(* IEC 61131-3 sources: Yaha/Documentation/Infomaterial/OSCAT/pcworx_building_100/pcworx_building_100/pcworx_building_100_module_export (part 2) *)

(* ---- TEMP_EXT.ST ---- *)
(*@PROPERTIES_EX@
TYPE: POU
LOCALE: 0
IEC_LANGUAGE: ST
PLC_TYPE: independent
PROC_TYPE: independent
GROUP: HLK
*)
(*@KEY@:DESCRIPTION*)
version 1.3	13. mar. 2009
programmer 	hugo
tested by	oscat

temp_ext measures and processes ext temperature and decides if heating or cooling is needed.

 the measurement of t_ext has 3 inputs which can be configured in different ways:
	t_ext_config = 0 means the ext temp is the avg of the 3 external temperatures, this mode is the default mode.
	t_ext_config = 1 means t_ext1 is used.
	t_ext_config = 2 means t_ext1 is used.
	t_ext_config = 3 means t_ext1 is used.
	t_ext_config = 4 means t_ext_default is used.
	t_ext_config = 5 means the lowest of the 3 external temperatures is used.
	t_ext_config = 6 means the higest externnal temperature is used.
	t_ext_config = 7 means the midlle external temperature is used, if there are only two working, the lowest is used.
	in any config mode, an external temperature higher then t_ext_max or lower then t_ext_min is ignored to prevent from temperatures caused by broken sensors or wires.
	if no external temperature is available, a default value (t_ext_default) is used.
	if you have only one external sensor, connect the 3 inputs to the same sensor, or select the right input with t_ext_config.

heating or cooling is enabled during heating / cooling period when the day or night start temperature is reached for at least the specified delay time and will be disabled after the stop temperature is reached.
t_ext output can be used by other modules to determine the correct system temperature for heating or cooling.
(*@KEY@:END_DESCRIPTION*)
FUNCTION_BLOCK TEMP_EXT

(*Group:Default*)

VAR_INPUT
	T_EXT1 :	REAL;
	T_EXT2 :	REAL;
	T_EXT3 :	REAL;
	T_EXT_CONFIG :	BYTE := 0;
	DT_IN :	UDINT;
	T_EXT_MIN :	REAL := REAL#-40.0;
	T_EXT_MAX :	REAL := REAL#60.0;
	T_EXT_DEFAULT :	REAL := REAL#-10.0;
	HEAT_PERIOD_START :	UDINT := UDINT#20995200;(*Anfangswert: D#1970-9-1*)
	HEAT_PERIOD_STOP :	UDINT := UDINT#10281600;(*Anfangswert: D#1970-4-30*)
	COOL_PERIOD_START :	UDINT := UDINT#07776000;(*Anfangswert: D#1970-4-1*)
	COOL_PERIOD_STOP :	UDINT := UDINT#23500800;(*Anfangswert: D#1970-9-30*)
	HEAT_START_TEMP_DAY :	REAL := REAL#15.0;
	HEAT_START_TEMP_NIGHT :	REAL := REAL#10.0;
	HEAT_STOP_TEMP :	REAL := REAL#18.0;
	COOL_START_TEMP_DAY :	REAL := REAL#26.0;
	COOL_START_TEMP_NIGHT :	REAL := REAL#26.0;
	COOL_STOP_TEMP :	REAL := REAL#24.0;
	START_DAY :	UDINT := UDINT#32400000;(*Anfangswert:TOD#09:00*)
	START_NIGHT :	UDINT := UDINT#75600000;(*Anfangswert:TOD#21:00*)
	CYCLE_TIME :	TIME := t#10m;
END_VAR

VAR_OUTPUT
	T_EXT :	REAL;
	HEAT :	BOOL;
	COOL :	BOOL;
END_VAR

VAR
	tx :	TIME;
	last_run :	TIME;
	init :	BOOL;
	cool_start :	UDINT;
	cool_stop :	UDINT;
	heat_start :	UDINT;
	heat_stop :	UDINT;
	xdate :	UDINT;
	day :	BOOL;
	T_PLC_MS :	T_PLC_MS;
END_VAR

(*@KEY@: WORKSHEET
NAME: TEMP_EXT
IEC_LANGUAGE: ST
*)
IF NOT init THEN
	init := TRUE;
	heat_start := SET_DATE(1972,MONTH_OF_DATE(heat_period_start),DAY_OF_MONTH(heat_period_start));
	heat_stop := SET_DATE(1972,MONTH_OF_DATE(heat_period_stop),DAY_OF_MONTH(heat_period_stop));
	cool_start := SET_DATE(1972,MONTH_OF_DATE(cool_period_start),DAY_OF_MONTH(cool_period_start));
	cool_stop := SET_DATE(1972,MONTH_OF_DATE(cool_period_stop),DAY_OF_MONTH(cool_period_stop));
END_IF;

(* read system time *)
T_PLC_MS();
tx:= UDINT_TO_TIME(T_PLC_MS.T_PLC_MS);

(* for efficiency exit isf this program has been executed less then 1min ago *)
IF tx - last_run < cycle_time THEN RETURN; END_IF;

(* calculate frequently used variables *)
xdate := SET_DATE(1972,MONTH_OF_DATE(DT_TO_DATE(dt_in)),DAY_OF_MONTH(DT_TO_DATE(dt_in)));
day := DT_TO_TOD(dt_in) >= start_day AND  DT_TO_TOD(dt_in) < start_night;

(* read the correct external temperature depending on the t_ext_config setting *)
t_ext := MULTI_IN(t_ext1, t_ext2, t_ext3, t_ext_default, t_ext_min, t_ext_max, t_ext_config);

(* dtermine heating *)
IF (heat_start <= heat_stop AND xdate >= heat_start AND xdate <= heat_stop) OR (heat_start > heat_stop AND (xdate >= heat_start OR xdate <= heat_stop)) THEN
	(* heating period id true check for temperature *)
	IF day AND t_ext <= heat_start_temp_day THEN
		heat := TRUE;
	ELSIF NOT day AND t_ext <= heat_start_temp_night THEN
		heat := TRUE;
	ELSIF t_ext >= heat_stop_temp THEN
		heat := FALSE;
	END_IF;
ELSE
	heat := FALSE;
END_IF;

(* dtermine cooling *)
IF (cool_start <= cool_stop AND xdate >= cool_start AND xdate <= cool_stop) OR (cool_start > cool_stop AND (xdate >= cool_start OR xdate <= cool_stop)) THEN
	(* cooling period is true check for temperature *)
	IF day AND t_ext >= cool_start_temp_day THEN
		cool := TRUE;
	ELSIF NOT day AND t_ext >= cool_start_temp_night THEN
		cool := TRUE;
	ELSIF t_ext <= cool_stop_temp THEN
		cool := FALSE;
	END_IF;
ELSE
	cool := FALSE;
END_IF;

last_run := tx;

(* revision history
hm	6 dec 2006	rev 1.0
	original version

hm	15.9.2007		rev 1.1
	replaced Time() with T_PLC_MS for compatibility and performance reasons

hm	7. oct. 2008	rev 1.2
	changed name of function month to month_of_date

hm	13. mar. 2009	rev 1.3
	real constants updated to new systax using dot

*)
(*@KEY@: END_WORKSHEET *)
END_FUNCTION_BLOCK

(* ---- TIMER_1.ST ---- *)
(*@PROPERTIES_EX@
TYPE: POU
LOCALE: 0
IEC_LANGUAGE: ST
PLC_TYPE: independent
PROC_TYPE: independent
GROUP: ELECTRICAL
*)
(*@KEY@:DESCRIPTION*)
version 2.2	16. dec. 2009
programmer 	oscat
tested by	oscat

this is a simple timer that generates an output pulse on selected days.
the output pulse width can be programmed with duration, if set to 0 no pulse is generated.
day specifies the specific days for the event to occur, bit 0 = sunday, bit 1 = saturday, bit 2 = friday ....
for all days to be active 127 has to be specified for DAY.
(*@KEY@:END_DESCRIPTION*)
FUNCTION_BLOCK TIMER_1

(*Group:Default*)

VAR_INPUT
	E :	BOOL := TRUE;
	DTI :	UDINT;
	START :	UDINT;
	DURATION :	TIME;
	DAY :	BYTE := BYTE#2#0111_1111;
END_VAR

VAR_OUTPUT
	Q :	BOOL;
	STOP :	TIME;
END_VAR

(*@KEY@: WORKSHEET
NAME: TIMER_1
IEC_LANGUAGE: ST
*)
IF E THEN
	stop := TOD_TO_TIME(START) + DURATION;
	IF stop > T#24h THEN stop := stop - T#24h; END_IF;
	Q := TIMECHECK(DT_TO_TOD(DTI), START, TIME_TO_TOD(stop)) AND (SHR(BYTE#128, DAY_OF_WEEK(DT_TO_DATE(DTI))) AND DAY) > BYTE#0;
ELSE
	Q := FALSE; (* clear output when e is not true *)
END_IF;

(*
1.12.2006 hm		rev 1.1
	corrected an error with pulse width = 0.

25.12.2006 hm		rev 1.2
	corrected an error when timer overflows.

14.apr 2007 hm		rev 1.3
	corrected an error while while output would not go active when start year would be 1970.
	increase accuracy by checking every 100ms
	added init section to compensate for timer overflow

15.9.2007 hm		rev 1.4
	replaced Time() with T_PLC_MS for compatibility and performance reasons

hm	1. okt 2007		rev 1.5
	corrected an error while output would not stay active over midnight.

hm	17. jan 2008	rev 1.6
	New code with better performance
	Output is now only active during the time of day it is supposed to
	no pulse is generated at power up

hm	7. oct. 2008	rev 1.7
	changed function weekday to day_of_week

hm	23. oct. 2008	rev 2.0
	new code, added input E, now days can be selected by bits in byte day

hm	6. nov. 2008	rev 2.1
	added default for input EN and input DAY

hm 16. dec 2009	rev 2.2
	fixed a bug over midnight

*)
(*@KEY@: END_WORKSHEET *)
END_FUNCTION_BLOCK

(* ---- TIMER_2.ST ---- *)
(*@PROPERTIES_EX@
TYPE: POU
LOCALE: 0
IEC_LANGUAGE: ST
PLC_TYPE: independent
PROC_TYPE: independent
GROUP: ELECTRICAL
*)
(*@KEY@:DESCRIPTION*)
version 1.5	22.dec.2008
programmer 	oscat
tested by	oscat

this timer generated programmabe output pulses per day, week, month and so on.
the mode input determines on which days the timer will be active.
	mode = 0			never
	mode = 1..7			monday .. sunday
	mode = 11			every day
	mode = 12			every second day
	mode = 13			every 3rd day
	mode = 14			every 4th day
	mode = 15			every 5th day
	mode = 16 			every 6th day
	mode = 20			only monday - friday
	mode = 21			only sat - sunday
	mode = 22			workdays only
	mode = 23			holidays and weekend
	mode = 24			holidays only
	mode = 25			every 1st day of the month
	mode = 26			every last day of the month
	mode = 27			every 31 of december
	mode = 28			every 1st of january

a holiday input can be used to supply holiday information to the module.
(*@KEY@:END_DESCRIPTION*)
FUNCTION_BLOCK TIMER_2

(*Group:Default*)

VAR_INPUT
	DT_IN :	UDINT;
	START :	UDINT;
	DURATION :	TIME;
	MODE :	BYTE;
	HOLIDAY :	BOOL;
END_VAR

VAR_OUTPUT
	Q :	BOOL;
END_VAR

VAR
	last_check :	TIME := T#0s;
	dat :	UDINT;
	daytime :	UDINT;
	activation :	TIME;
	tx :	TIME;
	enabled :	BOOL;
	wday :	INT;
	init :	BOOL;
END_VAR

VAR RETAIN
	run_date :	UDINT;
END_VAR

VAR
	T_PLC_MS :	T_PLC_MS;
END_VAR

(*@KEY@: WORKSHEET
NAME: TIMER_2
IEC_LANGUAGE: ST
*)
(* read system time *)
T_PLC_MS();
tx:= UDINT_TO_TIME(T_PLC_MS.T_PLC_MS);

IF NOT init THEN
	init := TRUE;
	last_check := tx - t#100ms;
END_IF;

(* for performance resons exit if execution is not necessary *)
IF tx - last_check < T#100ms THEN RETURN; END_IF;

(* calculate temp variables *)
dat := DT_TO_DATE(dt_in);
daytime := DT_TO_TOD(dt_in);
wday := DAY_OF_WEEK(dat);

(* calculate if any action is necessary today *)
CASE _BYTE_TO_INT(mode) OF
1..7:	(* mondays to fridays *)
	enabled := wday = _BYTE_TO_INT(mode);
11:	(* every day *)
	enabled := TRUE;
12..16:	(* every nth day *)
	enabled := (dat / UDINT#86400) MOD (BYTE_TO_UDINT(mode) - UDINT#10) = UDINT#0;
20:	(* monday - friday *)
	enabled := wday <= 5;
21:	(* saturday and sunday *)
	enabled := wday > 5;
22: (* workdays only *)
	enabled := wday <= 5 AND NOT holiday;
23:	(* holidays and weekends *)
	enabled := wday > 5 OR holiday;
24:	(* holidays only *)
	enabled := holiday;
25:	(* 1st day of the month *)
	enabled := DAY_OF_MONTH(dat) = 1;
26:	(* last day of month *)
	enabled := day_of_month(dat + TIME_TO_UDINT(t#1d)) = 1;
27:	(* 31st of december *)
	enabled := DAY_OF_MONTH(dat) = 31 AND MONTH_OF_DATE(dat) = 12;
28:	(* 1st of january *)
	enabled := DAY_OF_YEAR(dat) = 1;
ELSE
	enabled := FALSE;
END_CASE;

(* set output if necessary *)
IF enabled AND NOT Q AND daytime >= start AND run_date <> dat THEN
	Q := TRUE;
	activation := tx;
	run_date := dat;
ELSIF Q AND tx - activation >= duration THEN
	Q := FALSE;
END_IF;
last_check := Tx;

(* revision history
hm 22.2.2007		rev 1.1
	changed VAR RETAIN PERSISTENT to VAR RETAIN for better compatibility
	wago lon contollers do not support persisitent

hm	15.9.2007		rev 1.2
	replaced Time() with T_PLC_MS for compatibility and performance reasons

hm	7. oct. 2008	rev 1.3
	changed function month to month_of_date

hm	20. oct. 2008	rev 1.4
	improved performance
	deleted unnecessary trunc

hm	22. dec. 2008	rev 1.5
	make sure timer_2 is executed in the first cycle

*)
(*@KEY@: END_WORKSHEET *)
END_FUNCTION_BLOCK

(* ---- TIMER_EVENT_DECODE.ST ---- *)
(*@PROPERTIES_EX@
TYPE: POU
LOCALE: 0
IEC_LANGUAGE: ST
PLC_TYPE: independent
PROC_TYPE: independent
GROUP: ELECTRICAL
*)
(*@KEY@:DESCRIPTION*)
version 1.1	25. oct. 2008
programmer 	hugo
tested by	oscat

STRING_TO_TIMER_EVENT converts a string to a timer event structure.
(*@KEY@:END_DESCRIPTION*)
FUNCTION_BLOCK TIMER_EVENT_DECODE

(*Group:Default*)

VAR_INPUT
	EVENT :	oscat_STRING250;
	LANG :	INT;
END_VAR

VAR_OUTPUT
	TIMER_EVENT_DECODE :	oscat_TIMER_EVENT_DATA;
END_VAR

VAR
	pos :	INT;
	start :	INT;
	stop :	INT;
	step :	INT;
	tmp :	oscat_STRING60;
	char :	INT;
	FSTRING_TO_BYTE :	FSTRING_TO_BYTE;
	IS_CC :	IS_CC;
	FSTRING_TO_WEEK :	FSTRING_TO_WEEK;
	FSTRING_TO_WEEKDAY :	FSTRING_TO_WEEKDAY;
	STRING_TO_TOD :	STRING_TO_TOD;
	_STRING_TO_TIME :	_STRING_TO_TIME;
END_VAR

(*@KEY@: WORKSHEET
NAME: TIMER_EVENT_DECODE
IEC_LANGUAGE: ST
*)
(* a timer event is specified as follows:
	$typ;ch;day;start;duration;land;lor#
$ 		= start of definition
typ 	= type of definition	(number)
channel	= channel number		(number)
day 	= day number			(number)
start	= start time			(time of day)
duration= duration of event		(time)
land	= mask for output AND	(8bit value)
lor		= mask for ourput OR	(8bit value)
#		= end of definition
*)

(* check for start and ending character *)
stop := LEN(event);
IF (GET_CHAR(event,1) <> 60) AND (GET_CHAR(event,stop) <> 62) THEN RETURN; END_IF;
start := 2;
step := 0;

(* parse the string for next ; *)
FOR pos := 2 TO stop DO
    char := GET_CHAR(event,pos);

	IF char = 59 OR char = 62 THEN
		tmp := MID(event, pos - start, start);
		CASE step OF
			0:	(* read type *)
                FSTRING_TO_BYTE(IN:=tmp);
                TIMER_EVENT_DECODE.typ := FSTRING_TO_BYTE.FSTRING_TO_BYTE;

			1:	(* read channel *)
                FSTRING_TO_BYTE(IN:=tmp);
                TIMER_EVENT_DECODE.channel := FSTRING_TO_BYTE.FSTRING_TO_BYTE;

			2:	(* read day *)
                IS_CC(str:=tmp,cmp:='0123456789abcdefABCDEF#');

				IF IS_CC.IS_CC THEN
                    FSTRING_TO_BYTE(IN:=tmp);
                    TIMER_EVENT_DECODE.DAY := FSTRING_TO_BYTE.FSTRING_TO_BYTE;
				ELSIF TIMER_EVENT_DECODE.typ = BYTE#2 THEN
                    FSTRING_TO_WEEK(WEEK:=tmp,LANG:=LANG);
                    TIMER_EVENT_DECODE.DAY := FSTRING_TO_WEEK.FSTRING_TO_WEEK;
				ELSE
                    FSTRING_TO_WEEKDAY(WDAY:=tmp,LANG:=LANG);
                    TIMER_EVENT_DECODE.DAY := INT_TO_BYTE(FSTRING_TO_WEEKDAY.FSTRING_TO_WEEKDAY);
				END_IF;

			3:	(* read start *)
			    STRING_TO_TOD(_TOD:=tmp);
                TIMER_EVENT_DECODE.start := STRING_TO_TOD.STRING_TO_TOD;

			4:	(* read duaration *)
                _STRING_TO_TIME(_TIME:=tmp);
                TIMER_EVENT_DECODE.duration := _STRING_TO_TIME.STRING_TO_TIME;

			5:	(* read land *)
                FSTRING_TO_BYTE(IN:=tmp);
				TIMER_EVENT_DECODE.land := FSTRING_TO_BYTE.FSTRING_TO_BYTE;

			6:	(* read lor *)
                FSTRING_TO_BYTE(IN:=tmp);
				TIMER_EVENT_DECODE.LOR := FSTRING_TO_BYTE.FSTRING_TO_BYTE;
		END_CASE;
		start := pos + 1;
		step := step + 1;
	END_IF;
END_FOR;

(* revision history
hm	17. jun 2008	rev 1.0
	original version

hm	25. oct. 2008	rev 1.1
	adding input lang for language selection
*)
(*@KEY@: END_WORKSHEET *)
END_FUNCTION_BLOCK

(* ---- TIMER_EXT.ST ---- *)
(*@PROPERTIES_EX@
TYPE: POU
LOCALE: 0
IEC_LANGUAGE: ST
PLC_TYPE: independent
PROC_TYPE: independent
GROUP: ELECTRICAL
*)
(*@KEY@:DESCRIPTION*)
version 1.0	7. oct. 2008
programmer 	oscat
tested by	tobias

TIMER_EXT is a twilight timer.
the timer can be programmed to switch lights or other equippment or during twilight times.
in addition to the automatik mode the timer can be stopped and started by a switch at any given time.
An enable input ENA can be used for external control.
two inputs ON and OFF can be used to statically control the output.
the timer can be programmed to work on saturdays, sundays and holidays if required.
(*@KEY@:END_DESCRIPTION*)
FUNCTION_BLOCK TIMER_EXT

(*Group:Default*)

VAR_INPUT
	ENA :	BOOL;
	ON :	BOOL;
	OFF :	BOOL;
	MAN :	BOOL;
	SWITCH :	BOOL;
	DT_IN :	UDINT;
	SUN_SET :	UDINT;
	SUN_RISE :	UDINT;
	HOLIDAY :	BOOL;
	T_DEBOUNCE :	TIME := T#100ms;
	T_RISE_START :	TIME;
	T_RISE_STOP :	TIME;
	T_SET_START :	TIME;
	T_SET_STOP :	TIME;
	T_DAY_START :	UDINT;
	T_DAY_STOP :	UDINT;
	ENABLE_SATURDAY :	BOOL;
	ENABLE_SUNDAY :	BOOL;
	ENABLE_HOLIDAY :	BOOL;
END_VAR

VAR_OUTPUT
	Q :	BOOL;
	STATUS :	BYTE;
END_VAR

VAR
	mx :	MANUAL_2;
	deb :	DEBOUNCE;
	tdx :	UDINT;
	wdx :	INT;
	tc :	TIME;
	tx :	UDINT;
	tl :	UDINT;
	qx :	BOOL;
	T_PLC_MS :	T_PLC_MS;
	init :	BOOL;
END_VAR

(*@KEY@: WORKSHEET
NAME: TIMER_EXT
IEC_LANGUAGE: ST
*)
(* lösche die millisekunden bei sunrise und sunset *)
SUN_RISE := SUN_RISE / UDINT#1000 * UDINT#1000;
SUN_SET := SUN_SET / UDINT#1000 * UDINT#1000;

(* measure cycle time tc and make sure this circuitry is not called more then once in 200ms*)
T_PLC_MS();
tx:= T_PLC_MS.T_PLC_MS;
IF NOT init THEN
	init := TRUE;
	tl := tx;
END_IF;
tc := UDINT_TO_TIME(tx - tl);
IF tc < t#200ms THEN RETURN; END_IF;
tl := tx;

(* debounce *)
deb(in := SWITCH, TD := T_DEBOUNCE, PM := TRUE);

(* read time of day and strip off all milliseconds *)
tdx := DT_TO_TOD(dt_in);
wdx := DAY_OF_WEEK(DT_TO_DATE(dt_in));

(* automatic output control *)
IF deb.Q THEN
	qx := NOT qx;
	status := BYTE#110;
ELSIF holiday AND NOT enable_holiday THEN
	qx := FALSE;
ELSIF wdx = 6 AND NOT enable_saturday THEN
	qx := FALSE;
ELSIF wdx = 7 AND NOT enable_sunday THEN
	qx := FALSE;
ELSIF T_day_start > UDINT#00 (* TOD#00:00 *) AND tdx - T_DAY_START <= TIME_TO_UDINT(tc) THEN
	(* turn on at specified daytime *)
	qx := TRUE;
	status := BYTE#111;
ELSIF T_DAY_STOP > UDINT#00 (* TOD#00:00 *) AND tdx - T_DAY_STOP <= TIME_TO_UDINT(tc) THEN
	(* turn off at specific daytime *)
	qx := FALSE;
	status := BYTE#112;
ELSIF T_RISE_START > T#0s AND tdx - SUN_RISE + TIME_TO_UDINT(T_RISE_START) <= TIME_TO_UDINT(tc) THEN
	(* turn on before sunrise *)
	qx := TRUE;
	status := BYTE#113;
ELSIF T_RISE_STOP > T#0s AND tdx - SUN_RISE - TIME_TO_UDINT(T_RISE_STOP) <= TIME_TO_UDINT(tc) THEN
	(* turn off after sunrise *)
	qx := FALSE;
	status := BYTE#114;
ELSIF T_SET_start > T#0s AND tdx - SUN_SET + TIME_TO_UDINT(T_SET_START) <= TIME_TO_UDINT(tc) THEN
	(* turn on before sunset *)
	qx := TRUE;
	status := BYTE#115;
ELSIF T_SET_STOP > T#0s AND tdx - SUN_SET - TIME_TO_UDINT(T_SET_STOP) <= TIME_TO_UDINT(tc) THEN
	(* turn off after sunset *)
	qx := FALSE;
	status := BYTE#116;
END_IF;

(* manual and output control *)
mx(in := qx, ena := ENA, on := ON, off := OFF, man := MAN);
Q := mx.Q;

(* set the status output *)
IF mx.STATUS > BYTE#100 THEN status := mx.STATUS; END_IF;

(*
hm 7. oct. 2008	rev 1.0
	original version

*)
(*@KEY@: END_WORKSHEET *)
END_FUNCTION_BLOCK

(* ---- TIMER_P4.ST ---- *)
(*@PROPERTIES_EX@
TYPE: POU
LOCALE: 0
IEC_LANGUAGE: ST
PLC_TYPE: independent
PROC_TYPE: independent
GROUP: ELECTRICAL
*)
(*@KEY@:DESCRIPTION*)
version 1.4	26. jan. 2011
programmer 	hugo
tested by	oscat

TIMER_P4 is a programmable universal timer.
(*@KEY@:END_DESCRIPTION*)
FUNCTION_BLOCK TIMER_P4

(*Group:Default*)

VAR_INPUT
	DTIME :	UDINT;
	TREF_0 :	UDINT;
	TREF_1 :	UDINT;
	HOLY :	BOOL;
	L0 :	BOOL;
	L1 :	BOOL;
	L2 :	BOOL;
	L3 :	BOOL;
	OFS :	BYTE;
	ENQ :	BOOL;
	MAN :	BOOL;
	MI :	BYTE;
	RST :	BOOL;
END_VAR

VAR_IN_OUT
	PROG :	oscat_TIMER_EVENT;
END_VAR

VAR_OUTPUT
	Q0 :	BOOL;
	Q1 :	BOOL;
	Q2 :	BOOL;
	Q3 :	BOOL;
	STATUS :	BYTE;
END_VAR

VAR
	day_start :	UDINT;
	start :	UDINT;
	event :	oscat_TIMER_EVENT_DATA;
	pos :	INT;
	last_execute :	UDINT;
	current_day :	DINT;
	mask :	BYTE;
	ma :	oscat_arb_0_3;
	mo :	oscat_arb_0_3;
	qn :	oscat_TP4_qn;
	qs :	oscat_TP4_qn;
	channel :	INT;
	tx :	UDINT;
	array_max :	INT := 63;
	channel_max :	INT := 3;
END_VAR

(*@KEY@: WORKSHEET
NAME: TIMER_P4
IEC_LANGUAGE: ST
*)
(* for performance reasons we only execute the code at the beginning of a new second *)

IF RST THEN
	(* reset all events to last active on 1.1.1970 *)
	last_execute := UDINT#00; (* DT#1970-1-1-00:00 *)
	FOR pos := 0 TO ARRAY_MAX DO
		IF (PROG[pos].CHANNEL >= OFS) AND (_BYTE_TO_INT(PROG[pos].CHANNEL) < (_BYTE_TO_INT(OFS) + 4)) THEN PROG[pos].LAST := last_execute; END_IF;
	END_FOR;

	(* reset all set markers and logic masks *)
	FOR pos := 0 TO channel_max DO
		qs[pos] := FALSE;
	END_FOR;

(* normal operation *)
ELSIF dtime <> last_execute THEN
	(* save the actual second for next execution test *)
	last_execute := DTIME;

	(* calculate dt for the start of the day to be used in comparisons *)
	day_start := DATE_TO_DT(DT_TO_DATE(DTIME));

	(* set all qn to FALSE *)
	FOR pos := 0 TO channel_max DO qn[pos] := FALSE; END_FOR;

	(* search the array PROG for timer events *)
	FOR pos := 0 TO ARRAY_MAX DO
		event := prog[pos];
		channel := _BYTE_TO_INT(event.CHANNEL) - _BYTE_TO_INT(OFS);
		IF (event.TYP > BYTE#0) AND (channel >= 0) AND (channel <= channel_max) THEN
			ma[channel] := event.LAND;
			mo[channel] := event.LOR;
			CASE _BYTE_TO_INT(event.TYP) OF
				1:	(* daily event *)
					start := day_start + event.start;
					qn[channel] := dtime >= start AND dtime <= start + TIME_TO_UDINT(event.DURATION);

				2: 	(* event by selected weekdays *)
					IF (SHR(BYTE#128, DAY_OF_WEEK(DT_TO_DATE(Dtime))) AND event.DAY) > BYTE#0 THEN
						start := day_start + event.start;
						qn[channel] := dtime >= start AND dtime <= start + TIME_TO_UDINT(event.DURATION);
					END_IF;

				3:	(* event every N days *)
					IF current_day MOD _BYTE_TO_DINT(event.DAY) = DINT#0 THEN
						start := day_start + event.start;
						qn[channel] := dtime >= start AND dtime <= start + TIME_TO_UDINT(event.DURATION);
					END_IF;

				10:	(* weekly event exactly once a week the weekday is specified in day, 1= mo *)
					IF DAY_OF_WEEK(DT_TO_DATE(DTIME)) = BYTE_TO_INT(event.DAY) THEN
						start := day_start + event.start;
						qn[channel] := dtime >= start AND dtime <= start + TIME_TO_UDINT(event.DURATION);
					END_IF;

				20:	(* monthly event *)
					IF DAY_OF_MONTH(DT_TO_DATE(DTIME)) = BYTE_TO_INT(event.DAY) THEN
						start := day_start + event.start;
						qn[channel] := dtime >= start AND dtime <= start + TIME_TO_UDINT(event.DURATION);
					END_IF;

				21:	(* event on last day of month *)
					IF DT_TO_DATE(DTIME) = MONTH_END(DT_TO_DATE(dtime)) THEN
						start := day_start + event.start;
						qn[channel] := dtime >= start AND dtime <= start + TIME_TO_UDINT(event.DURATION);
					END_IF;

				30:	(* yearly event on a specific day specified in day *)
					IF DAY_OF_YEAR(DT_TO_DATE(DTIME)) = BYTE_TO_INT(event.DAY) THEN
						start := day_start + event.start;
						qn[channel] := dtime >= start AND dtime <= start + TIME_TO_UDINT(event.DURATION);
					END_IF;

				31:	(* event on last day of year *)
					IF DT_TO_DATE(DTIME) = YEAR_END(YEAR_OF_DATE(DT_TO_DATE(dtime))) THEN
						start := day_start + event.start;
						qn[channel] := dtime >= start AND dtime <= start + TIME_TO_UDINT(event.DURATION);
					END_IF;

				40:	(* event on leap days *)
					IF LEAP_DAY(DT_TO_DATE(dtime)) THEN
						start := day_start + event.start;
						qn[channel] := dtime >= start AND dtime <= start + TIME_TO_UDINT(event.DURATION);
					END_IF;

				41: (* event on holidays *)
					IF HOLY THEN
						start := day_start + event.start;
						qn[channel] := dtime >= start AND dtime <= start + TIME_TO_UDINT(event.DURATION);
					END_IF;

				42: (* event on holidays and weekends *)
					IF (Holy OR (DAY_OF_WEEK(DT_TO_DATE(dtime)) = 6) OR (DAY_OF_WEEK(DT_TO_DATE(dtime)) = 7)) THEN
						start := day_start + event.start;
						qn[channel] := dtime >= start AND dtime <= start + TIME_TO_UDINT(event.DURATION);
					END_IF;

				43:	(* event on workdays Mo-FR and no holiday *)
					IF DAY_OF_WEEK(DT_TO_DATE(dtime)) < 6 THEN
						start := day_start + event.start;
						qn[channel] := dtime >= start AND dtime <= start + TIME_TO_UDINT(event.DURATION);
					END_IF;

				50: (* event after reference time *)
					CASE _BYTE_TO_INT(prog[pos].DAY) OF
						0:	tx := tref_0;
						1:	tx := tref_1;
					ELSE
						tx := UDINT#0 (* TOD#00:00 *);
					END_CASE;
					start := day_start + tx + event.start;
					qn[channel] := dtime >= start AND dtime <= start + TIME_TO_UDINT(event.DURATION);

				51:	(* event before reference time *)
					CASE _BYTE_TO_INT(prog[pos].DAY) OF
						0:	tx := tref_0;
						1:	tx := tref_1;
					ELSE
						tx := UDINT#0 (* TOD#00:00 *);
					END_CASE;
					start := day_start + tx - event.start;
					qn[channel] := dtime >= start AND dtime <= start + TIME_TO_UDINT(event.DURATION);

				52 : (* set output at specific time + offset  *)
					CASE _BYTE_TO_INT(prog[pos].DAY) OF
						0:	tx := tref_0;
						1:	tx := tref_1;
					ELSE
						tx := UDINT#0 (* TOD#00:00 *);
					END_CASE;
					start := day_start + tx + event.start;
					IF dtime >= start AND day_start > event.LAST THEN
						qs[channel] := TRUE;
						prog[pos].LAST := day_start;
					END_IF;

				53 : (* reset output at specific time + offset *)
					CASE _BYTE_TO_INT(prog[pos].DAY) OF
						0:	tx := tref_0;
						1:	tx := tref_1;
					ELSE
						tx := UDINT#0 (* TOD#00:00 *);
					END_CASE;
					start := day_start + tx + event.start;
					IF dtime >= start AND day_start > event.LAST THEN
						qs[channel] := FALSE;
						prog[pos].LAST := day_start;
					END_IF;

				54 : (* set output at specific time - offset  *)
					CASE _BYTE_TO_INT(prog[pos].DAY) OF
						0:	tx := tref_0;
						1:	tx := tref_1;
					ELSE
						tx := UDINT#0 (* TOD#00:00 *);
					END_CASE;
					start := day_start + tx - event.start;
					IF dtime >= start AND day_start > event.LAST THEN
						qs[channel] := TRUE;
						prog[pos].LAST := day_start;
					END_IF;

				55 : (* reset output at specific time - offset *)
					CASE _BYTE_TO_INT(prog[pos].DAY) OF
						0:	tx := tref_0;
						1:	tx := tref_1;
					ELSE
						tx := UDINT#0 (* TOD#00:00 *);
					END_CASE;
					start := day_start + tx - event.start;
					IF dtime >= start AND day_start > event.LAST THEN
						qs[channel] := FALSE;
						prog[pos].LAST := day_start;
					END_IF;
			END_CASE;
		END_IF;
	END_FOR;
END_IF;

(* prepare the logical input mask *)
mask := BYTE#255;
mask:=BIT_LOAD_B(mask,L0,0);
mask:=BIT_LOAD_B(mask,L1,1);
mask:=BIT_LOAD_B(mask,L2,2);
mask:=BIT_LOAD_B(mask,L3,3);

(* set the outputs *)
Q0 := ENQ AND ((qn[0] OR qs[0]) AND ((ma[0] AND mask) = ma[0]) OR ((mo[0] AND mask) > BYTE#0) OR (man AND BIT_OF_DWORD(BYTE_TO_DWORD(MI),0)));
Q1 := ENQ AND ((qn[1] OR qs[1]) AND ((ma[1] AND mask) = ma[1]) OR ((mo[1] AND mask) > BYTE#1) OR (man AND BIT_OF_DWORD(BYTE_TO_DWORD(MI),1)));
Q2 := ENQ AND ((qn[2] OR qs[2]) AND ((ma[2] AND mask) = ma[2]) OR ((mo[2] AND mask) > BYTE#2) OR (man AND BIT_OF_DWORD(BYTE_TO_DWORD(MI),2)));
Q3 := ENQ AND ((qn[3] OR qs[3]) AND ((ma[3] AND mask) = ma[3]) OR ((mo[3] AND mask) > BYTE#3) OR (man AND BIT_OF_DWORD(BYTE_TO_DWORD(MI),3)));

(* set status *)
IF NOT enq THEN
	status := BYTE#100;
ELSIF man THEN
	status := BYTE#101;
ELSE
	status := BYTE#102;
END_IF;

(* revision history
hm	17. jun 2008	rev 1.0
	original version

hm	9. oct. 2008	rev 1.1
	changed function year to year_of_date
	changed function weekday to day_of_week
	changed structure of program to be more efficient
	changed input DIS to ENQ

hm	18. oct. 2008	rev 1.2
	changed type of input OFS from int to byte
	added typecasts to avoid warnings

hm	28. feb. 2009	rev 1.3
	array was not correctly initialized

hm	26. jan 2011	rev 1.4
	changed code to allow events over midnight
*)
(*@KEY@: END_WORKSHEET *)
END_FUNCTION_BLOCK

(* ---- WATER_CP.ST ---- *)
(*@PROPERTIES_EX@
TYPE: POU
LOCALE: 0
IEC_LANGUAGE: ST
PLC_TYPE: independent
PROC_TYPE: independent
GROUP: HLK
*)
(*@KEY@:DESCRIPTION*)
version 1.2	13. mar. 2009
programmer 	hugo
tested by	tobias

water_cp calculates the specific heat capacity of liquid water from 0..100 °C
(*@KEY@:END_DESCRIPTION*)
FUNCTION_BLOCK WATER_CP

(*Group:Default*)

VAR_INPUT
	T :	REAL;
END_VAR

VAR_OUTPUT
	CAP :	REAL;
END_VAR

VAR
	Pts :	INT;
	data :	oscat_XY;
	FB_LINEAR_INT :	LINEAR_INT;
END_VAR

(*@KEY@: WORKSHEET
NAME: WATER_CP
IEC_LANGUAGE: ST
*)
IF Pts = 0 THEN
    Pts := 10;

    data[01][0] := REAL#0.0;
    data[01][1] := REAL#4.228;
    data[02][0] := REAL#05.0;
    data[02][1] := REAL#4.200;
    data[03][0] := REAL#10.0;
    data[03][1] := REAL#4.188;
    data[04][0] := REAL#15.0;
    data[04][1] := REAL#4.184;
    data[05][0] := REAL#50.0;
    data[05][1] := REAL#4.181;
    data[06][0] := REAL#60.0;
    data[06][1] := REAL#4.183;
    data[07][0] := REAL#70.0;
    data[07][1] := REAL#4.187;
    data[08][0] := REAL#80.0;
    data[08][1] := REAL#4.194;
    data[09][0] := REAL#90.0;
    data[09][1] := REAL#4.204;
    data[10][0] := REAL#100.0;
    data[10][1] := REAL#4.220;

END_IF;

FB_LINEAR_INT(X:=T,XY:=Data,Pts:=Pts);
cap:=FB_LINEAR_INT.LINEAR_INT;

(*
    °C - die Celsius-Temperatur in Grad Celsius
    v – das spezifische Volumen in Kubikdezimeter je Kilogramm dm³/kg
    h – die spezifische Enthalpie in Kilojoule je Kilogramm 	kJ/kg
    u – die spezifische Innere Energie in Kilojoule je Kilogramm 	kJ/kg
    s – die spezifische Entropie in Kilojoule je Kilogramm mal Kelvin 	kJ/(kg·K)
    cp - die spezifische Wärmekapazität bei konstantem Druck in Kilojoule je Kilogramm mal Kelvin 	kJ/(kg·K)
    Y – Volumenausdehnungskoeffizient in 10-3 durch Kelvin  10-3/K
    L – Wärmeleitfähigkeit in Milliwatt je Meter mal Kelvin  mW / (m·K)
    n – Viskosität in Mikropascal mal Sekunde uPa·s
    s ? – Oberflächenspannung in Millinewton je Meter  mN/m

°C 		v 				h 			u 		s 			cp 		Y 		L		n		s
-20		1,006580
0 		1,000160 		0,06 		-0,04 	-0,0001 	4,228 	-0,080 	561,0 	1792 	75,65
4		1,000028
5 		1,0000 		21,1 		21,0 	0,076 		4,200 	0,011 	570,6 	1518 	74,95
10 		1,0003 		42,1 		42,0 	0,151 		4,188 	0,087 	580,0 	1306 	74,22
15 		1,0009 		63,0 		62,9 	0,224 		4,184 	0,152 	589,4 	1137 	73,49
20 		1,001797 		83,9 		83,8 	0,296 		4,183 	0,209 	598,4 	1001 	72,74
25 		1,0029 		104,8 		104,7 	0,367 		4,183 	0,259 	607,2 	890,4 	71,98
30 		1,0044 		125,8 		125,7 	0,437 		4,183 	0,305 	615,5 	797,7 	71,20
35 		1,0060 		146,7 		146,6 	0,505 		4,183 	0,347 	623,3 	719,6 	70,41
40 		1,007842 		167,58 	167,5 	0,572 		4,182 	0,386 	630,6 	653,3 	69,60
45 		1,0099 		188,5 		188,4 	0,638 		4,182 	0,423 	637,3 	596,3 	68,78
50 		1,0121 		209,4 		209,3 	0,704 		4,181 	0,457 	643,6 	547,1 	67,95
60 		1,017089 		251,2 		251,1 	0,831 		4,183 	0,522 	654,4 	466,6 	66,24
70 		1,0227 		293,1 		293,0 	0,955 		4,187 	0,583 	663,1 	404,1 	64,49
80 		1,029027 		335,0 		334,9 	1,075 		4,194 	0,640 	670,0 	354,5 	62,68
90 		1,0359 		377,0 		376,9 	1,193 		4,204 	0,696 	675,3 	314,6 	60,82
99,63 	1,0431 		417,5 		417,4 	1,303 		4,217 	0,748 	679,0 	283,0 	58,99
100	1,043453		419,1

Stoffdaten von Wasser Quelle Wickipedia

Wasser hat unter Normaldruck seine größte Dichte von 1000 Kilogramm pro Kubikmeter bei 3,98 °C und zeigt damit eine Dichteanomalie.
Diese besteht darin, dass sich Wasser unterhalb von 3,98 °C bei weiterer Temperaturverringerung, auch beim Wechsel zum festen
Aggregatzustand, wieder ausdehnt, was man nur von wenigen Stoffen kennt. Die derzeit genauesten publizierten Werte für die maximale
Dichte liegen bei (999,974950 ± 0,00084) kg/m³ und bei (3,983 ± 0,00067) °C für die Temperatur, bei der dieser Wert erreicht wird.
Die Werte stellen einen Mittelwert der von verschiedenen physikalischen Instituten veröffentlichten Zahlen dar (Stand 2001).

Die Berechnung der Dichte von luftfreiem Wasser DLF in Abhängigkeit von der Temperatur T ([T] = °C) kann mit Hilfe der folgenden
Virialgleichung erfolgen:
: \frac{D_{\rm LF}}{\rm g/l} = \frac{a_0 + a_1 T + a_2 T^2 + a_3 T^3 + a_4 T^4 + a_5 T^5}{1 + b T}.
mit den Koeffizienten: a0 = 999,83952; a1 = 16,952577 (°C)-1; a2 = -7,9905127·10-3 (°C)-2; a3 = -4,6241757·10-5 (°C)-3;
a4 = 1,0584601·10-7 (°C)-4; a5 = -2,8103006·10-10 (°C)-5 und b = 0,0168872.
Für die Berechnung der Dichte von luftgesättigtem Wasser korrigiert man den Wert nach
DLG/(g/l) = DLF/(g/l) - 0,004612 + 0,000106 (°C)-1·T. (Quelle: PTB-Mitteilungen 100/3-90)

*)

(* revision history

hm	29.10.2007	rev 1.0
	original version

hm	27. dec 2007	rev 1.1
	increased accuracy

hm	13. mar. 2009	rev 1.2
	real constants updated to new systax using dot

*)
(*@KEY@: END_WORKSHEET *)
END_FUNCTION_BLOCK

(* ---- WATER_ENTHALPY.ST ---- *)
(*@PROPERTIES_EX@
TYPE: POU
LOCALE: 0
IEC_LANGUAGE: ST
PLC_TYPE: independent
PROC_TYPE: independent
GROUP: HLK
*)
(*@KEY@:DESCRIPTION*)
version 1.1	13. mar. 2009
programmer 	hugo
tested by	tobias

water_enthalpy calculates the enthalpy of liquid water from 0..100 °C
(*@KEY@:END_DESCRIPTION*)
FUNCTION_BLOCK WATER_ENTHALPY

(*Group:Default*)

VAR_INPUT
	T :	REAL;
END_VAR

VAR_OUTPUT
	RESULT :	REAL;
END_VAR

VAR
	Pts :	INT;
	data :	oscat_XY;
	FB_LINEAR_INT :	LINEAR_INT;
END_VAR

(*@KEY@: WORKSHEET
NAME: WATER_ENTHALPY
IEC_LANGUAGE: ST
*)
IF Pts = 0 THEN
    Pts := 11;
    data[01][0] := REAL#0.0;
    data[01][1] := REAL#0.06;
    data[02][0] := REAL#10.0;
    data[02][1] := REAL#42.1;
    data[03][0] := REAL#20.0;
    data[03][1] := REAL#83.9;
    data[04][0] := REAL#30.0;
    data[04][1] := REAL#125.8;
    data[05][0] := REAL#40.0;
    data[05][1] := REAL#167.58;
    data[06][0] := REAL#50.0;
    data[06][1] := REAL#209.4;
    data[07][0] := REAL#60.0;
    data[07][1] := REAL#251.2;
    data[08][0] := REAL#70.0;
    data[08][1] := REAL#293.1;
    data[09][0] := REAL#80.0;
    data[09][1] := REAL#335.0;
    data[10][0] := REAL#90.0;
    data[10][1] := REAL#377.0;
    data[11][0] := REAL#100.0;
    data[11][1] := REAL#419.1;
END_IF;

FB_LINEAR_INT(X:=T,XY:=Data,Pts:=Pts);
Result :=FB_LINEAR_INT.LINEAR_INT;

(*
    °C - die Celsius-Temperatur in Grad Celsius
    v – das spezifische Volumen in Kubikdezimeter je Kilogramm dm³/kg
    h – die spezifische Enthalpie in Kilojoule je Kilogramm 	kJ/kg
    u – die spezifische Innere Energie in Kilojoule je Kilogramm 	kJ/kg
    s – die spezifische Entropie in Kilojoule je Kilogramm mal Kelvin 	kJ/(kg·K)
    cp - die spezifische Wärmekapazität bei konstantem Druck in Kilojoule je Kilogramm mal Kelvin 	kJ/(kg·K)
    Y – Volumenausdehnungskoeffizient in 10-3 durch Kelvin  10-3/K
    L – Wärmeleitfähigkeit in Milliwatt je Meter mal Kelvin  mW / (m·K)
    n – Viskosität in Mikropascal mal Sekunde uPa·s
    s ? – Oberflächenspannung in Millinewton je Meter  mN/m

°C 		v 				h 			u 		s 			cp 		Y 		L		n		s
-20		1,006580
0 		1,000160 		0,06 		-0,04 	-0,0001 	4,228 	-0,080 	561,0 	1792 	75,65
4		1,000028
5 		1,0000 		21,1 		21,0 	0,076 		4,200 	0,011 	570,6 	1518 	74,95
10 		1,0003 		42,1 		42,0 	0,151 		4,188 	0,087 	580,0 	1306 	74,22
15 		1,0009 		63,0 		62,9 	0,224 		4,184 	0,152 	589,4 	1137 	73,49
20 		1,001797 		83,9 		83,8 	0,296 		4,183 	0,209 	598,4 	1001 	72,74
25 		1,0029 		104,8 		104,7 	0,367 		4,183 	0,259 	607,2 	890,4 	71,98
30 		1,0044 		125,8 		125,7 	0,437 		4,183 	0,305 	615,5 	797,7 	71,20
35 		1,0060 		146,7 		146,6 	0,505 		4,183 	0,347 	623,3 	719,6 	70,41
40 		1,007842 		167,58 	167,5 	0,572 		4,182 	0,386 	630,6 	653,3 	69,60
45 		1,0099 		188,5 		188,4 	0,638 		4,182 	0,423 	637,3 	596,3 	68,78
50 		1,0121 		209,4 		209,3 	0,704 		4,181 	0,457 	643,6 	547,1 	67,95
60 		1,017089 		251,2 		251,1 	0,831 		4,183 	0,522 	654,4 	466,6 	66,24
70 		1,0227 		293,1 		293,0 	0,955 		4,187 	0,583 	663,1 	404,1 	64,49
80 		1,029027 		335,0 		334,9 	1,075 		4,194 	0,640 	670,0 	354,5 	62,68
90 		1,0359 		377,0 		376,9 	1,193 		4,204 	0,696 	675,3 	314,6 	60,82
99,63 	1,0431 		417,5 		417,4 	1,303 		4,217 	0,748 	679,0 	283,0 	58,99
100	1,043453		419,1

Stoffdaten von Wasser Quelle Wickipedia

Wasser hat unter Normaldruck seine größte Dichte von 1000 Kilogramm pro Kubikmeter bei 3,98 °C und zeigt damit eine Dichteanomalie.
Diese besteht darin, dass sich Wasser unterhalb von 3,98 °C bei weiterer Temperaturverringerung, auch beim Wechsel zum festen
Aggregatzustand, wieder ausdehnt, was man nur von wenigen Stoffen kennt. Die derzeit genauesten publizierten Werte für die maximale
Dichte liegen bei (999,974950 ± 0,00084) kg/m³ und bei (3,983 ± 0,00067) °C für die Temperatur, bei der dieser Wert erreicht wird.
Die Werte stellen einen Mittelwert der von verschiedenen physikalischen Instituten veröffentlichten Zahlen dar (Stand 2001).

Die Berechnung der Dichte von luftfreiem Wasser DLF in Abhängigkeit von der Temperatur T ([T] = °C) kann mit Hilfe der folgenden
Virialgleichung erfolgen:
: \frac{D_{\rm LF}}{\rm g/l} = \frac{a_0 + a_1 T + a_2 T^2 + a_3 T^3 + a_4 T^4 + a_5 T^5}{1 + b T}.
mit den Koeffizienten: a0 = 999,83952; a1 = 16,952577 (°C)-1; a2 = -7,9905127·10-3 (°C)-2; a3 = -4,6241757·10-5 (°C)-3;
a4 = 1,0584601·10-7 (°C)-4; a5 = -2,8103006·10-10 (°C)-5 und b = 0,0168872.
Für die Berechnung der Dichte von luftgesättigtem Wasser korrigiert man den Wert nach
DLG/(g/l) = DLF/(g/l) - 0,004612 + 0,000106 (°C)-1·T. (Quelle: PTB-Mitteilungen 100/3-90)

*)

(* revision history
hm	13. mar. 2009	rev 1.0
	original version

hm	13. mar. 2009	rev 1.1
	real constants updated to new systax using dot

*)
(*@KEY@: END_WORKSHEET *)
END_FUNCTION_BLOCK

(* ---- AIR_DENSITY.ST ---- *)
(*@PROPERTIES_EX@
TYPE: POU
LOCALE: 0
IEC_LANGUAGE: ST
PLC_TYPE: independent
PROC_TYPE: independent
GROUP: HLK
*)
(*@KEY@:DESCRIPTION*)
version 1.3	13. mar. 2009
programmer 	hugo
tested by	tobias

this function calculates the air density between 0 and 100 deg C
(*@KEY@:END_DESCRIPTION*)
FUNCTION AIR_DENSITY:REAL

(*Group:Default*)

VAR_INPUT
	T :	REAL;
	P :	REAL;
	RH :	REAL;
END_VAR

(*@KEY@: WORKSHEET
NAME: AIR_DENSITY
IEC_LANGUAGE: ST
*)
AIR_DENSITY := 101325.0 * (1.0 - RH * SDD(T, TRUE) * 3.773319E-3 / P) / (287.05 * ( T - -273.15));

(* original code used for rev 1.0

SDD := SDD(T,FALSE);
RF := RL / (1- RH*SDD/P*RX);
Air_density := P / (RF * (T-TK));

*)

(* revision history

hm	29.10.2007	rev 1.0
	original version

hm	4.12.2007		rev 1.1
	changed code for better performance

hm	18. oct. 2008	rev 1.2
	using phys constants

hm	13. mar. 2009	rev 1.3
	real constants updated to new systax using dot

*)
(*@KEY@: END_WORKSHEET *)
END_FUNCTION

(* ---- AIR_ENTHALPY.ST ---- *)
(*@PROPERTIES_EX@
TYPE: POU
LOCALE: 0
IEC_LANGUAGE: ST
PLC_TYPE: independent
PROC_TYPE: independent
GROUP: HLK
*)
(*@KEY@:DESCRIPTION*)
version 1.0	31 oct 2007
programmer 	hugo
tested by	tobias

this function calculates the enthalpy for humid air between 0 and 100 deg C
(*@KEY@:END_DESCRIPTION*)
FUNCTION AIR_ENTHALPY:REAL

(*Group:Default*)

VAR_INPUT
	T :	REAL;
	RH :	REAL;
END_VAR

(*@KEY@: WORKSHEET
NAME: AIR_ENTHALPY
IEC_LANGUAGE: ST
*)
Air_enthalpy := 1.00482 * T + (1.86 * T + 2500.78) * dew_con(RH,T);

(* revision history

hm	31.10.2007		rev 1.0
	original version

hm	2.11.2007		rev 1.1
	deleted unused variable RF

hm	2.12.2007		rev 1.2
	changed code for better performance
*)
(*@KEY@: END_WORKSHEET *)
END_FUNCTION

(* ---- BUILDING_VERSION.ST ---- *)
(*@PROPERTIES_EX@
TYPE: POU
LOCALE: 0
IEC_LANGUAGE: ST
PLC_TYPE: independent
PROC_TYPE: independent
GROUP: OTHER
*)
(*@KEY@:DESCRIPTION*)
version 1.1	16 dec 2007
programmer 	hugo
tested by	tobias

oscat_version returns the version number in dword format
132 is library version 1.32
if IN = true, the release date will be returned
(*@KEY@:END_DESCRIPTION*)
FUNCTION BUILDING_VERSION:DWORD

(*Group:Default*)

VAR_INPUT
	IN :	BOOL;
END_VAR

(*@KEY@: WORKSHEET
NAME: BUILDING_VERSION
IEC_LANGUAGE: ST
*)
IF in THEN
	BUILDING_VERSION := UDINT_TO_DWORD(set_Date(2011,02,03));
ELSE
	BUILDING_VERSION := DWORD#100;
END_IF;

(* revision history
hm	6. oct 2006	rev 1.0
	original version

hm	16. dec 2007	rev 1.1
	added possibility to return date and version depending on IN.

*)

(*@KEY@: END_WORKSHEET *)
END_FUNCTION

(* ---- DEW_CON.ST ---- *)
(*@PROPERTIES_EX@
TYPE: POU
LOCALE: 0
IEC_LANGUAGE: ST
PLC_TYPE: independent
PROC_TYPE: independent
GROUP: HLK
*)
(*@KEY@:DESCRIPTION*)
version 1.6	19. jan. 2011
programmer 	hugo
tested by	oscat

this function calculates the water concentratin in air for a given temperature and relative humidity.
the output states the concentration of water vapor in air in Gramms / qubic meter.
(*@KEY@:END_DESCRIPTION*)
FUNCTION DEW_CON:REAL

(*Group:Default*)

VAR_INPUT
	RH :	REAL;
	T :	REAL;
END_VAR

(*@KEY@: WORKSHEET
NAME: DEW_CON
IEC_LANGUAGE: ST
*)
(*	this code is good to read but need to be improoved
	SDD := 6.1078*EXPT(10,(a*T)/(b+T));
	DD := RH/100 * SDD;
	V := LOG(DD/6.1078);
	TD := b*V/(a-v);
	dew_con := 0.1 * mw / RU * DD / (T - TK);
*)
IF RH > 0.0 AND T > -50.0 THEN
	DEW_CON := 2.166824303E-2 * RH * SDD(T,FALSE)  / (T - -273.15);
ELSE
	DEW_CON := 0.0;
END_IF;

(*
Bezeichnungen:
r = relative Luftfeuchte
T = Temperatur in °C
TK = Temperatur in Kelvin (TK = T + 273.15)
TD = Taupunkttemperatur in °C
DD = Dampfdruck in hPa
SDD = Sättigungsdampfdruck in hPa

Parameter:
a = 7.5, b = 237.3 für T >= 0
a = 7.6, b = 240.7 für T < 0 über Wasser (Taupunkt)
a = 9.5, b = 265.5 für T < 0 über Eis (Frostpunkt)

R* = 8314.3 J/(kmol*K) (universelle Gaskonstante)
mw = 18.016 kg (Molekulargewicht des Wasserdampfes)
AF = absolute Feuchte in g Wasserdampf pro m3 Luft

Formeln:

   1. SDD(T) = 6.1078 * 10^((a*T)/(b+T))
   2. DD(r,T) = r/100 * SDD(T)
   3. r(T,TD) = 100 * SDD(TD) / SDD(T)
   4. TD(r,T) = b*v/(a-v) mit v(r,T) = log10(DD(r,T)/6.1078)
   5. AF(r,TK) = 10^5 * mw/R* * DD(r,T)/TK; AF(TD,TK) = 10^5 * mw/R* * SDD(TD)/TK

*)

(* revision history

hm 29 apr 2007	rev 1.0
	original version

hm	13.sep 2007	rev 1.1
	improoved coding for speed
	deleted unused variabled SDD,DD,V, TD

hm	2. dec 2007	rev 1.2
	changed code for better performance
	output is now in Gramms / Qubic meter

hm	14. oct. 2008	rev 1.3
	performance improvement

hm	18. oct. 2008	rev 1.4
	using phys constants

hm	13. mar. 2009	rev 1.5
	improved code

hm	19. jan. 2011	rev 1.6
	return value 0.0 if RH <= 0.0

*)
(*@KEY@: END_WORKSHEET *)
END_FUNCTION

(* ---- DEW_RH.ST ---- *)
(*@PROPERTIES_EX@
TYPE: POU
LOCALE: 0
IEC_LANGUAGE: ST
PLC_TYPE: independent
PROC_TYPE: independent
GROUP: HLK
*)
(*@KEY@:DESCRIPTION*)
version 1.2	13. mar. 2009
programmer 	hugo
tested by	tobias

this function calculates the relative humidity in air for a given temperature in °C and vapor concentration in Kg/m³..
(*@KEY@:END_DESCRIPTION*)
FUNCTION DEW_RH:REAL

(*Group:Default*)

VAR_INPUT
	VC :	REAL;
	T :	REAL;
END_VAR

(*@KEY@: WORKSHEET
NAME: DEW_RH
IEC_LANGUAGE: ST
*)
DEW_RH := LIMIT(0.0, VC / DEW_CON(1.0, T), 100.0);

(* code before rev 1.1
dew_rh := VC / dew_con(100,T) * 100;
IF dew_rh > 100 THEN dew_rh := 100; END_IF;
*)

(* revision history
hm	29. apr 2007	rev 1.0
	original version

hm	2. 12. 2007	rev 1.1
	new code for better performance

hm	13. mar. 2009	rev 1.2
	real constants updated to new systax using dot

*)
(*@KEY@: END_WORKSHEET *)
END_FUNCTION

(* ---- DEW_TEMP.ST ---- *)
(*@PROPERTIES_EX@
TYPE: POU
LOCALE: 0
IEC_LANGUAGE: ST
PLC_TYPE: independent
PROC_TYPE: independent
GROUP: HLK
*)
(*@KEY@:DESCRIPTION*)
version 1.6	13. mar. 2009
programmer 	hugo
tested by	oscat

this function calculates the dew point for air given the temperature and relative humidity.
dew_temp(60,0.25) = 16.7 °C.
which means the dew point for air with 25° and 60% RH is at 16.7 °C.
(*@KEY@:END_DESCRIPTION*)
FUNCTION DEW_TEMP:REAL

(*Group:Default*)

VAR_INPUT
	RH :	REAL;
	T :	REAL;
END_VAR

VAR
	V :	REAL;
END_VAR

(*@KEY@: WORKSHEET
NAME: DEW_TEMP
IEC_LANGUAGE: ST
*)
IF rh > 0.0 THEN
(*	old code was rewritten for better performance
	SDD := 6.1078*EXPT(10,(7.5*T)/(237.3+T));
	DD := RH/100 * SDD;
	V := LOG(DD/6.1078);
	dew_temp := 237.3*V/(7.5-v);
*)
	V := LOG(RH * 0.01 * EXP10((7.5*T) / (237.3+T)));
	DEW_TEMP := 237.3*V / (7.5-V);
ELSE
	DEW_TEMP:= -273.15;
END_IF;

(* revision history

hm		2.10.2006	rev 1.0
	original version created

hm		29.4.2007	rev 1.1
	checked for rh not to be 0 because log(0) is not defined

hm		13.9.2007	rev 1.2
	code rewritten for better performance

hm	2. dec 2007	rev 1.3
	changed code for better performance

hm	8. jan 2008	rev 1.4
	further improvement in performance

hm	18. oct. 2008	rev 1.5
	using phys constants

hm	13. mar. 2009	rev 1.6
	real constants updated to new systax using dot

*)

(*
Bezeichnungen:
r = relative Luftfeuchte
T = Temperatur in °C
TK = Temperatur in Kelvin (TK = T + 273.15)
TD = Taupunkttemperatur in °C
DD = Dampfdruck in hPa
SDD = Sättigungsdampfdruck in hPa

Parameter:
a = 7.5, b = 237.3 für T >= 0
a = 7.6, b = 240.7 für T < 0 über Wasser (Taupunkt)
a = 9.5, b = 265.5 für T < 0 über Eis (Frostpunkt)

R* = 8314.3 J/(kmol*K) (universelle Gaskonstante)
mw = 18.016 kg (Molekulargewicht des Wasserdampfes)
AF = absolute Feuchte in g Wasserdampf pro m3 Luft

Formeln:

   1. SDD(T) = 6.1078 * 10^((a*T)/(b+T))
   2. DD(r,T) = r/100 * SDD(T)
   3. r(T,TD) = 100 * SDD(TD) / SDD(T)
   4. TD(r,T) = b*v/(a-v) mit v(r,T) = log10(DD(r,T)/6.1078)
   5. AF(r,TK) = 10^5 * mw/R* * DD(r,T)/TK; AF(TD,TK) = 10^5 * mw/R* * SDD(TD)/TK

*)
(*@KEY@: END_WORKSHEET *)
END_FUNCTION

(* ---- HEAT_INDEX.ST ---- *)
(*@PROPERTIES_EX@
TYPE: POU
LOCALE: 0
IEC_LANGUAGE: ST
PLC_TYPE: independent
PROC_TYPE: independent
GROUP: HLK
*)
(*@KEY@:DESCRIPTION*)
version 1.3	13. mar. 2009
programmer 	hugo
tested by	tobias

this function calculates the heat index temperature depending on external temperature and Relative humidity
(*@KEY@:END_DESCRIPTION*)
FUNCTION HEAT_INDEX:REAL

(*Group:Default*)

VAR_INPUT
	T :	REAL;
	RH :	REAL;
END_VAR

VAR
	RH2 :	REAL;
	T2 :	REAL;
	TX :	REAL;
END_VAR

(*@KEY@: WORKSHEET
NAME: HEAT_INDEX
IEC_LANGUAGE: ST
*)
IF RH < 20.0 OR T < 20.0 THEN
	HEAT_INDEX := T;
ELSE
	TX := T;
	RH2 := RH * RH;
	TX := C_TO_F(TX);
	T2 := TX * TX;
	HEAT_INDEX := -42.379 + 2.04901523 * TX - 6.83783E-3 * T2
			+ RH * (10.1433127 - 0.22475541 * TX + 1.22874E-3 * T2)
			+ RH2 * (8.5282E-4 * TX - 5.481717E-2 - 1.99E-6 * T2);
	HEAT_INDEX := F_TO_C(HEAT_INDEX);
END_IF;

(* revision history

hm 27.2.2007		rev 1.1
	deleted unused variables rh3 and T3

hm	2.12.2007		rev 1.2
	changed code for better performance

hm	13. mar. 2009	rev 1.3
	real constants updated to new systax using dot

*)
(*@KEY@: END_WORKSHEET *)
END_FUNCTION

(* ---- SDD.ST ---- *)
(*@PROPERTIES_EX@
TYPE: POU
LOCALE: 0
IEC_LANGUAGE: ST
PLC_TYPE: independent
PROC_TYPE: independent
GROUP: HLK
*)
(*@KEY@:DESCRIPTION*)
version 1.1	2 dec 2007
programmer 	hugo
tested by	tobias

this function calculates the vapor saturation pressure for moist Air over ice or water
(*@KEY@:END_DESCRIPTION*)
FUNCTION SDD:REAL

(*Group:Default*)

VAR_INPUT
	T :	REAL;
	ICE :	BOOL;
END_VAR

(*@KEY@: WORKSHEET
NAME: SDD
IEC_LANGUAGE: ST
*)
IF ice THEN
	SDD := 611.153 * EXP(22.4433 * T / (272.186 + T));
ELSE
	SDD := 611.213 * EXP(17.5043 * T / (241.2 + T));
END_IF;

(* old code used in rev 1.0
IF ice THEN
	SDD := 611.153 * exp10(9.747*T / (272.186 + T));
ELSE
	SDD := 611.213 * exp10(7.602*T / (241.2 + T));
END_IF;
*)

(* revision history

hm 29 oct 2007		rev 1.0
	original version

hm	2. dec 2007		rev 1.1
	changed code for better performance
*)
(*@KEY@: END_WORKSHEET *)
END_FUNCTION

(* ---- SDD_NH3.ST ---- *)
(*@PROPERTIES_EX@
TYPE: POU
LOCALE: 0
IEC_LANGUAGE: ST
PLC_TYPE: independent
PROC_TYPE: independent
GROUP: HLK
*)
(*@KEY@:DESCRIPTION*)
version 1.0	19 Aug 2009
programmer 	hugo
tested by	tobias

this function calculates the vapor saturation pressure for NH3 gas
valid input temperature range is -109°C .. 98 °C
(*@KEY@:END_DESCRIPTION*)
FUNCTION SDD_NH3:REAL

(*Group:Default*)

VAR_INPUT
	T :	REAL;
END_VAR

(*@KEY@: WORKSHEET
NAME: SDD_NH3
IEC_LANGUAGE: ST
*)
(*
calculate according to NIST
Antoine Equation Parameters
log10(P) = A - (B / (T + C))
	P = vapor pressure (bar)
	T = temperature (K)
Temperature (K)	A	B	C	Reference	Comment

 T = 164.0 - 239.5, A =	3.18757, B =506.713, C=-80.78	Stull, 1947	Coefficents calculated by NIST from author's data.
 T = 239.5 - 371.4, A =	4.86886, B = 1113.928, C = -10.409	Stull, 1947	Coefficents calculated by NIST from author's data.
*)

IF T < -33.65 THEN
	SDD_NH3 := EXP(7.3396511649 - ( 1166.7498002 / ( T + 192.37 )));
ELSE
	SDD_NH3 := EXP(11.210964456 - ( 2564.9140075 / ( T + 262.741 )));
END_IF;

(* revision history

hm 19 aug 2009		rev 1.0
	original version

*)
(*@KEY@: END_WORKSHEET *)
END_FUNCTION

(* ---- SDT_NH3.ST ---- *)
(*@PROPERTIES_EX@
TYPE: POU
LOCALE: 0
IEC_LANGUAGE: ST
PLC_TYPE: independent
PROC_TYPE: independent
GROUP: HLK
*)
(*@KEY@:DESCRIPTION*)
version 1.0	20 Aug 2009
programmer 	hugo
tested by	tobias

this function calculates the vapor saturation temperature for NH3 gas
valid input pressure is 0.001 bar .. 60 bar.
(*@KEY@:END_DESCRIPTION*)
FUNCTION SDT_NH3:REAL

(*Group:Default*)

VAR_INPUT
	P :	REAL;
END_VAR

(*@KEY@: WORKSHEET
NAME: SDT_NH3
IEC_LANGUAGE: ST
*)
(*
calculate according to NIST
Antoine Equation Parameters
log10(P) = A - (B / (T + C))
	P = vapor pressure (bar)
	T = temperature (K)
Temperature (K)	A	B	C	Reference	Comment

 T = 164.0 - 239.5, A =	3.18757, B =506.713, C=-80.78	Stull, 1947	Coefficents calculated by NIST from author's data.
 T = 239.5 - 371.4, A =	4.86886, B = 1113.928, C = -10.409	Stull, 1947	Coefficents calculated by NIST from author's data.
*)

IF P < 1.0E-3 THEN
	SDT_NH3 := -110.0;
ELSIF P < 1.0 THEN
	SDT_NH3 := 506.713 / (3.18757 - LOG(P)) - 192.37 ;
ELSE
	SDT_NH3 := 1113.928 / (4.86886 - LOG(P)) - 262.71 ;
END_IF;

(* revision history

hm 20 aug 2009		rev 1.0
	original version

*)
(*@KEY@: END_WORKSHEET *)
END_FUNCTION

(* ---- TANK_VOL1.ST ---- *)
(*@PROPERTIES_EX@
TYPE: POU
LOCALE: 0
IEC_LANGUAGE: ST
PLC_TYPE: independent
PROC_TYPE: independent
GROUP: HLK
*)
(*@KEY@:DESCRIPTION*)
version 1.0	10. Mar 2010
programmer 	hugo
tested by	tobias

TANK_VOL1 calculates the volume of a tubular tank filled to level H.
(*@KEY@:END_DESCRIPTION*)
FUNCTION TANK_VOL1:REAL

(*Group:Default*)

VAR_INPUT
	TR :	REAL;
	TL :	REAL;
	H :	REAL;
END_VAR

(*@KEY@: WORKSHEET
NAME: TANK_VOL1
IEC_LANGUAGE: ST
*)
TANK_VOL1 := CIRCLE_SEG(TR, H) * TL;

(* revision histroy
hm	10. mar 2010	rev 1.0
	original version

*)
(*@KEY@: END_WORKSHEET *)
END_FUNCTION

(* ---- TANK_VOL2.ST ---- *)
(*@PROPERTIES_EX@
TYPE: POU
LOCALE: 0
IEC_LANGUAGE: ST
PLC_TYPE: independent
PROC_TYPE: independent
GROUP: HLK
*)
(*@KEY@:DESCRIPTION*)
version 1.0	10. Mar 2010
programmer 	hugo
tested by	tobias

TANK_VOL2 calculates the volume of a spherical tank filled to level H.
(*@KEY@:END_DESCRIPTION*)
FUNCTION TANK_VOL2:REAL

(*Group:Default*)

VAR_INPUT
	TR :	REAL;
	H :	REAL;
END_VAR

(*@KEY@: WORKSHEET
NAME: TANK_VOL2
IEC_LANGUAGE: ST
*)
TANK_VOL2 := 3.14159265358979323846264338327950288 * H * H * (TR - H / 3.0);

(* revision histroy
hm	10. mar 2010	rev 1.0
	original version

*)
(*@KEY@: END_WORKSHEET *)
END_FUNCTION

(* ---- WATER_DENSITY.ST ---- *)
(*@PROPERTIES_EX@
TYPE: POU
LOCALE: 0
IEC_LANGUAGE: ST
PLC_TYPE: independent
PROC_TYPE: independent
GROUP: HLK
*)
(*@KEY@:DESCRIPTION*)
version 1.2	13. mar. 2009
programmer 	hugo
tested by	tobias

this function calculates the water density for air free water between 0 and 100 deg C
while sat is false the denisty is calculated for air free water and when sat = true
the calculation is performed for water saturated with air.
(*@KEY@:END_DESCRIPTION*)
FUNCTION WATER_DENSITY:REAL

(*Group:Default*)

VAR_INPUT
	T :	REAL;
	SAT :	BOOL;
END_VAR

VAR
	T2 :	REAL;
	T4 :	REAL;
END_VAR

(*@KEY@: WORKSHEET
NAME: WATER_DENSITY
IEC_LANGUAGE: ST
*)
T2 := T * T;
T4 := T2 * T2;
WATER_DENSITY := (999.83952 + 16.952577*T + -7.9905127E-3*T2 + -4.6241757E-5*T2*T + 1.0584601E-7*T4 + -2.8103006E-10*T4*T) / (1.0 + 0.0168872*T);
IF sat THEN WATER_DENSITY := WATER_DENSITY - 0.004612 + 0.000106 * T; END_IF;

(* revision history

hm	13.9.2007		rev 1.0
	original version

hm	2.12.2007		rev 1.1
	changed code for better performance

hm	13. mar. 2009	rev 1.2
	real constants updated to new systax using dot

*)

(*
    °C - die Celsius-Temperatur in Grad Celsius
    v – das spezifische Volumen in Kubikdezimeter je Kilogramm dm³/kg
    h – die spezifische Enthalpie in Kilojoule je Kilogramm 	kJ/kg
    u – die spezifische Innere Energie in Kilojoule je Kilogramm 	kJ/kg
    s – die spezifische Entropie in Kilojoule je Kilogramm mal Kelvin 	kJ/(kg·K)
    cp - die spezifische Wärmekapazität bei konstantem Druck in Kilojoule je Kilogramm mal Kelvin 	kJ/(kg·K)
    Y – Volumenausdehnungskoeffizient in 10-3 durch Kelvin  10-3/K
    L – Wärmeleitfähigkeit in Milliwatt je Meter mal Kelvin  mW / (m·K)
    n – Viskosität in Mikropascal mal Sekunde uPa·s
    s ? – Oberflächenspannung in Millinewton je Meter  mN/m

°C 		v 				h 			u 		s 			cp 		Y 		L		n		s
-20		1,006580
0 		1,000160 		0,06 		-0,04 	-0,0001 	4,228 	-0,080 	561,0 	1792 	75,65
4		1,000028
5 		1,0000 		21,1 		21,0 	0,076 		4,200 	0,011 	570,6 	1518 	74,95
10 		1,0003 		42,1 		42,0 	0,151 		4,188 	0,087 	580,0 	1306 	74,22
15 		1,0009 		63,0 		62,9 	0,224 		4,184 	0,152 	589,4 	1137 	73,49
20 		1,001797 		83,9 		83,8 	0,296 		4,183 	0,209 	598,4 	1001 	72,74
25 		1,0029 		104,8 		104,7 	0,367 		4,183 	0,259 	607,2 	890,4 	71,98
30 		1,0044 		125,8 		125,7 	0,437 		4,183 	0,305 	615,5 	797,7 	71,20
35 		1,0060 		146,7 		146,6 	0,505 		4,183 	0,347 	623,3 	719,6 	70,41
40 		1,007842 		167,58 	167,5 	0,572 		4,182 	0,386 	630,6 	653,3 	69,60
45 		1,0099 		188,5 		188,4 	0,638 		4,182 	0,423 	637,3 	596,3 	68,78
50 		1,0121 		209,4 		209,3 	0,704 		4,181 	0,457 	643,6 	547,1 	67,95
60 		1,017089 		251,2 		251,1 	0,831 		4,183 	0,522 	654,4 	466,6 	66,24
70 		1,0227 		293,1 		293,0 	0,955 		4,187 	0,583 	663,1 	404,1 	64,49
80 		1,029027 		335,0 		334,9 	1,075 		4,194 	0,640 	670,0 	354,5 	62,68
90 		1,0359 		377,0 		376,9 	1,193 		4,204 	0,696 	675,3 	314,6 	60,82
99,63 	1,0431 		417,5 		417,4 	1,303 		4,217 	0,748 	679,0 	283,0 	58,99
100	1,043453		419,1

Stoffdaten von Wasser Quelle Wickipedia

*)
(*@KEY@: END_WORKSHEET *)
END_FUNCTION

(* ---- WCT.ST ---- *)
(*@PROPERTIES_EX@
TYPE: POU
LOCALE: 0
IEC_LANGUAGE: ST
PLC_TYPE: independent
PROC_TYPE: independent
GROUP: HLK
*)
(*@KEY@:DESCRIPTION*)
version 1.2	13. mar. 2009
programmer 	hugo
tested by	tobias

this function calculates the wind chill temperature
(*@KEY@:END_DESCRIPTION*)
FUNCTION WCT:REAL

(*Group:Default*)

VAR_INPUT
	T :	REAL;
	V :	REAL;
END_VAR

(*@KEY@: WORKSHEET
NAME: WCT
IEC_LANGUAGE: ST
*)
IF V < 5.0 OR T > 10.0 THEN
	WCT := T;
ELSE
	WCT := 13.12 + 0.6215 * T +(0.3965 * T - 11.37) * EXP(LN(v) * 0.16);
END_IF;

(* revision history
hm	7 feb 2007		rev 1.0
	original version

hm	7 dec 2007	rev 1.1
	changed code for better performance

hm	13. mar. 2009	rev 1.2
	real constants updated to new systax using dot

*)
(*@KEY@: END_WORKSHEET *)
END_FUNCTION
